PROGRAM MAIN
VAR
END_VAR

END_PROGRAM

(* stored: Version 1.1.0.1, ProductVersion 3.1.4024.4
   POU MAIN: Id {b852e6b0-fc65-4fe2-a4d1-3c982f793d34}, SpecialFunc None *)
